FUNCTION Get_PID_Gain : bool
VAR_INPUT
END_VAR
VAR
END_VAR

GVL.fbCoEReadP_X(
		Axis :=GVL.AxisX,		
		NetId := '5.33.182.40.1.1', 
  		Index := 16#3100,
  		pDstBuf := ADR(GVL.X_GetP_Gain), 
  		BufLen := SIZEOF(GVL.X_GetP_Gain), 
  		Execute := GVL.X_CoERead_EX, 
  		Timeout := T#1S, 	
	);	
GVL.fbCoEReadD_X(
		Axis :=GVL.AxisX,		
		NetId := '5.33.182.40.1.1', 
  		Index := 16#3101,
  		pDstBuf := ADR(GVL.X_GetD_Gain), 
  		BufLen := SIZEOF(GVL.X_GetD_Gain), 
  		Execute := GVL.X_CoERead_EX, 
  		Timeout := T#1S, 	
		
	);	
GVL.fbCoEReadI_X(
		Axis :=GVL.AxisX,		
		NetId := '5.33.182.40.1.1', 
  		Index := 16#3102,
  		pDstBuf := ADR(GVL.X_GetI_Gain), 
  		BufLen := SIZEOF(GVL.X_GetI_Gain), 
  		Execute := GVL.X_CoERead_EX, 
  		Timeout := T#1S, 	
	);	
GVL.X_CoERead_EX := FALSE;
	
GVL.fbCoEReadP_Y(
		Axis :=GVL.AxisY,		
		NetId := '5.33.182.40.1.1', 
  		Index := 16#3100,
  		pDstBuf := ADR(GVL.Y_GetP_Gain), 
  		BufLen := SIZEOF(GVL.Y_GetP_Gain), 
  		Execute := GVL.Y_CoERead_EX, 
  		Timeout := T#1S, 	
	);	
GVL.fbCoEReadD_Y(
		Axis :=GVL.AxisY,		
		NetId := '5.33.182.40.1.1', 
  		Index := 16#3101,
  		pDstBuf := ADR(GVL.Y_GetD_Gain), 
  		BufLen := SIZEOF(GVL.Y_GetD_Gain), 
  		Execute := GVL.Y_CoERead_EX, 
  		Timeout := T#1S, 	
		
	);	
GVL.fbCoEReadI_Y(
		Axis :=GVL.AxisY,		
		NetId := '5.33.182.40.1.1', 
  		Index := 16#3102,
  		pDstBuf := ADR(GVL.Y_GetI_Gain), 
  		BufLen := SIZEOF(GVL.X_GetI_Gain), 
  		Execute := GVL.Y_CoERead_EX, 
  		Timeout := T#1S, 	
	);	
GVL.Y_CoERead_EX := FALSE;

END_FUNCTION

(* stored: Version 1.1.0.1, ProductVersion 3.1.4024.12
   POU Get_PID_Gain: Id {2d4b600f-bed5-4753-8c95-a2b8d2aec812}, SpecialFunc None *)
